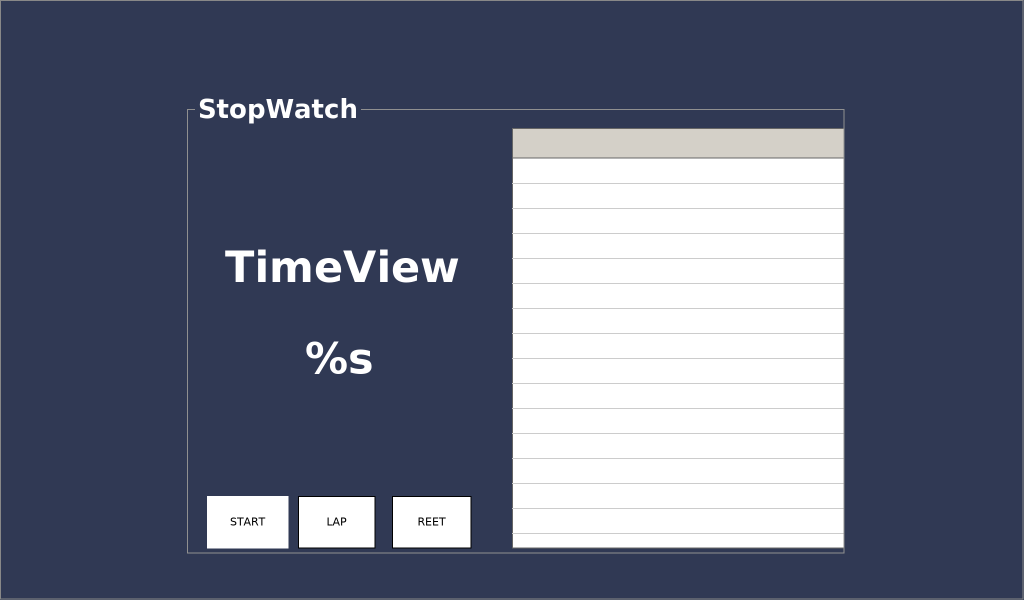
VISUALIZATION Main_views  // 1024x600
    Textfield (177,305 325x107), "%s", text variable: MAIN.FormattedTime
    Table (512,128 332x420), data array: MAIN.FormattedIntervals
        p3854506369: MAIN.FormattedIntervals[INDEX]
        p1014161805: 20 - 1 + INT#1
    Textfield (214,218 257x98), "TimeView"
    RoundedRectangle (207,496 81x52), "PAUSE", invisible if: NOT(MAIN.Timer.Running)
        tap MAIN.PauseButton
    RoundedRectangle (392,496 79x52), "REET"
        tap MAIN.ResetButton
    RoundedRectangle (298,496 77x52), "LAP", text variable: MAIN.IntervalButton
        tap MAIN.IntervalButton
    RoundedRectangle (207,496 81x52), "START", invisible if: MAIN.Timer.Running
        tap MAIN.StartButton
    Textfield (120,26 768x105)
    GroupBox (187,101 657x452), "StopWatch"
END_VISUALIZATION

(* stored: Version 1.1.0.1, ProductVersion 3.1.4026.8
   Visu Main_views: Id {4e292f34-e9a3-474a-b97e-3cd14fc5d717} *)
